{attribute 'qualified_only'}
TYPE E_LogSeverity_Ish :
(
	Info := ADSLOG_MSGTYPE_HINT,
	Warning := ADSLOG_MSGTYPE_WARN,
	Error := ADSLOG_MSGTYPE_ERROR
) DWORD;
END_TYPE

(* stored: Version 1.1.0.1, ProductVersion 3.1.4022.18
   DUT E_LogSeverity_Ish: Id {0e6a13b7-47f6-4a79-a023-1c2ce1af75ef} *)
